PROGRAM MAIN
VAR

init:BOOL;

uw1_Toque AT %I* 	: INT;
uw1_Position AT %I* 	: DINT;
TriggerOff:Trigger;
TriggerEM_Button:Trigger;
END_VAR


IF init =FALSE THEN
	init:=TRUE;
	ACT_Init_param();
END_IF

ACT_Emergency();

ACT_IO();

ACT_fbCall();

ACTION ACT_Emergency:

IF gMachineCtrl.Cmd.EmStop THEN
	//FB_Machine_Ctrl.ResetCycle:=TRUE;
	//gMachineCtrl.Cmd.EmStop:=FALSE;
	
	gMachineCtrl.Cmd.SwitchOn:=FALSE;
END_IF
IF TriggerOff.EDGENEG(gMachineCtrl.Cmd.SwitchOn) THEN
	gMachineCtrl.Cmd.EmStop:=TRUE;
END_IF

IF TriggerEM_Button.EDGEPOS(gMachineCtrl.Cmd.EmStop) THEN
	gMachineCtrl.Cmd.EmStop:=TRUE;
END_IF
END_ACTION

ACTION ACT_fbCall:



RwInverter(
	//Set_Vel_Link:=gUVCtrl.Input.Par.UV_Inverter_Set_Speed , 
	//INV_Enable:=gUVCtrl.Input.Cmd.UV_Inverter_Run , 
	//HWlink:=gMachineCtrl.IO.RwInverter,
	ctrl:=gMachineCtrl.RwInverter,
	//ResetError:= , 
	MasterNetId:= , 
	nSlaveAddr:= , 
	nSubIndex:= , 
	nIndex:= , 
	//Actual_Vel_Link=>gUVCtrl.Output.Status.UV_Inverter_Actual_Speed , 
	Error=> , 
	ErrorCode=> , 
	Inv_Status=> );


	
FB_OFF.Ctrl_ref 			REF= gMachineCtrl;
FB_OFF.FB_Machine_Run_ref 	REF= FB_Machine_Run;
FB_OFF.FB_Mechinit_ref 		REF= FB_Mechinit;
FB_OFF();	
	
FB_Machine_Ctrl.Ctrl_ref 				REF= gMachineCtrl;
FB_Machine_Ctrl.FB_Machine_Run_ref 		REF= FB_Machine_Run;
FB_Machine_Ctrl.FB_Mechinit_ref 		REF= FB_Mechinit;
FB_Machine_Ctrl.FB_MechinitOutput_ref  	REF= FB_Mechinit_Output;
FB_Machine_Ctrl.FB_OFF_ref				REF= FB_OFF;
FB_Machine_Ctrl();

FB_Machine_Run.Ctrl_ref 		REF= gMachineCtrl;
FB_Machine_Run.FB_RW_Ctrl_ref	REF= FB_RW_Ctrl;
FB_Machine_Run();


FB_Mechinit.Ctrl_ref	REF= gMachineCtrl;
FB_Mechinit();


FB_Mechinit_Output.Ctrl_ref	REF= gMachineCtrl;
FB_Mechinit_Output();

//FB_RW_Ctrl.Ctrl_ref REF= gMachineCtrl;
//FB_RW_Ctrl();
END_ACTION

ACTION ACT_Init_param:

//	Dancer fill speed
gMachineCtrl.Parameters.DancerFillSpeed:= 90000;//[mil deg/sec]

gMachineCtrl.Parameters.NumberOfCycles:= 1;

//Motor Parmeters
//gMachineCtrl.Parameters.MotorVelocity:=600;//[rpm]
gMachineCtrl.Parameters.DistanceToMove:=1000;//[mm]


gMachineCtrl.Parameters.WebLinarSpeed:=350;//[mm/sec]
gMachineCtrl.Parameters.WebLinarSpeedSlow:=250;//[mm/sec]

gMachineCtrl.Parameters.UW_1_Param.ForcedDiameter:=400;//[mm/sec]
gMachineCtrl.Parameters.UW_2_Param.ForcedDiameter:=400;//[mm/sec]

gMachineCtrl.Parameters.UW_1_Param.SetTension := 150;
gMachineCtrl.Parameters.UW_2_Param.SetTension := 150;

gMachineCtrl.Parameters.UW_1_Param.kp:=0.1;
gMachineCtrl.Parameters.UW_1_Param.TN:=T#0MS;

gMachineCtrl.Parameters.UW_2_Param.kp:=0.1;
gMachineCtrl.Parameters.UW_2_Param.TN:=T#0MS;

gMachineCtrl.Parameters.UW_1_Param.kpMove:=1;
gMachineCtrl.Parameters.UW_1_Param.TNMove:=T#0MS;

gMachineCtrl.Parameters.UW_2_Param.kpMove:=1;
gMachineCtrl.Parameters.UW_2_Param.TNMove:=T#0MS;
END_ACTION

ACTION ACT_IO:


//IO
gMachineCtrl.IO.In.PrimeryPressFeedback(
	SimFlag:= gMachineCtrl.Simulation);
	
gMachineCtrl.IO.In.SeconderyPressFeedbak(
	SimFlag:= gMachineCtrl.Simulation);
	
gMachineCtrl.IO.In.E_StopPressed := NOT(gMachineCtrl.IO.In.E_StopPressedRaw);
END_ACTION

END_PROGRAM

(* stored: Version 1.1.0.1, ProductVersion 3.1.4024.3
   POU MAIN: Id {906fbf26-856d-4f0f-b127-1015c6c2feda}, SpecialFunc None
   Action ACT_Emergency: Id {f209a312-0d75-4adb-886d-eb1e7339d1b2}
   Action ACT_fbCall: Id {82ef3718-f64a-421e-be71-e37b12e669fa}
   Action ACT_Init_param: Id {5ed366ef-f6c6-4a4b-b0fb-fb6ba19d4db9}
   Action ACT_IO: Id {2a18bd5c-a292-4da3-a0fd-3fbf174fcec3} *)
